PROGRAM gravarConfigPosicao021
VAR
	bReator: ARRAY[0..2] OF BOOL;
	posicaoAtual: STRING;
	enviaLog: STRING;
	estufaAtual: STRING;
END_VAR


// VERIFICA SE HA REATOR E MUDA A COR DO QUADRADO ------------------------------------
IF bReator[2] THEN
	gvl_p.aPositionsE021[gvl.actPos].cor:= 1;
	gvl_p.bCarrinhoReator3:=TRUE;
	gvl.cfgPos_Reat021:=TRUE;
	ELSE
		gvl_p.aPositionsE021[gvl.actPos].cor:=2;
		gvl_p.bCarrinhoReator3:=FALSE;
		gvl.cfgPos_Reat021:=FALSE;
END_IF

// REGISTRA AS INFORMAÇÕES EM CADA POSIÇÃO -------------------------------------------------------------
FOR gvl.n:=1 TO 24 BY 1 DO
	IF gvl.actPos = gvl.n THEN
		gvl_p.aPositionsE021[gvl.n].numOF:= gvl.cfgPos_OF021;
		gvl_p.aPositionsE021[gvl.n].lote:= gvl.cfgPos_LT021;
		gvl_p.aPositionsE021[gvl.n].class:= gvl.cfgPos_Class021;
		gvl_p.aPositionsE021[gvl.n].pot:= gvl.cfgPos_Pot021;
		gvl_p.aPositionsE021[gvl.n].reator:= gvl.cfgPos_Reat021;
		gvl_p.aPositionsE021[gvl.n].text:= insert(gvl.cfgPos_OF021,'-',5);
		gvl_p.aPositionsE021[gvl.n].text:= concat(gvl_p.aPositionsE021[gvl.n].text,gvl.cfgPos_LT021);
	END_IF
END_FOR

// DEFINIÇÃO DOS TEMPOS DE ACORDO COM AS CLASSES ----------------------------------------------
IF gvl_p.aPositionsE021[gvl.actPos].class <= 15 THEN
		GVL_p.arrStatusEstufas[2].tempoSecagem := T#60H;
		GVL_p.arrStatusEstufas[2].tempoArmazenagem := T#192H;
		gvl.totalSeca[2]:= '60';
		gvl_p.arrStatusEstufas[2].tempSeca:= 120;
		gvl.totalArm[2]:= '192';
		gvl_p.arrStatusEstufas[2].tempArm:= 70;
		ELSIF gvl_p.aPositionsE021[gvl.actPos].class > 15 THEN
			GVL_p.arrStatusEstufas[2].tempoSecagem:= T#96H;
			GVL_p.arrStatusEstufas[2].tempoArmazenagem:= T#240H;
			gvl.totalSeca[2]:= '96';
			gvl_p.arrStatusEstufas[2].tempSeca:= 120;
			gvl.totalArm[2]:= '240';
			gvl_p.arrStatusEstufas[2].tempArm:= 70;
END_IF

gvl.totalPos[2]:= gvl.totalPos[2] + 1;

///// GERADOR DE LOG -------------------------------------------------------------

posicaoAtual:= INT_TO_STRING(gvl.actPos);
estufaAtual:= INT_TO_STRING(gvl.actEst);
envialog:= 'Posição Nº ';
enviaLog:= concat(envialog, posicaoAtual);
enviaLog:= concat(envialog,' gravada.  ESTUFA 021');
gvl.logRegister19:= envialog;

END_PROGRAM

(* stored: Version 1.1.0.1, ProductVersion 3.1.4024.12
   POU gravarConfigPosicao021: Id {aaafc287-5d33-452c-add1-f546db79064b}, SpecialFunc None *)
